// TIA Portal V20 export
// export: Created 2025-12-01T14:57:26.6006718Z, ExportSetting None, DisplayName Totally Integrated Automation Portal, DisplayVersion V20 Update 3, DisplayName TIA Portal Openness, DisplayVersion V20 Update 3, DisplayName TIA Portal Version Control Interface, DisplayVersion V20 Update 3, DisplayName STEP 7 Professional, DisplayVersion V20 Update 3, DisplayName STEP 7 Safety, DisplayVersion V20 Update 2, DisplayName WinCC Basic/Comfort/Advanced, DisplayVersion V20 Update 3, DisplayName WinCC Professional, DisplayVersion V20 Update 3, DisplayName WinCC Unified, DisplayVersion V20 Update 3
FUNCTION "FC601_AJUSTE_SORTER_NEW" : Void   // FC601, LAD
{ S7_Optimized_Access := 'FALSE' }
// stored: AutoNumber false, SetENOAutomatically false
   VAR_INPUT
      Dato_encoder : DInt;
      Detector_referencia : Bool;
      activar_ajuste : Bool;
   END_VAR
   VAR_IN_OUT
      maux_fp_ajuste : Bool;
      maux_fp_detector : Bool;
      primer_flanco : DInt;
      segundo_flanco : DInt;
      tercer_flanco : DInt;
      cuarto_flanco : DInt;
      fin_medicion : Bool;
   END_VAR
   VAR_TEMP   // added for the SCL form of the ladder/FBD networks
      _w1 : Bool;
      _w2 : Bool;
   END_VAR
BEGIN

REGION Network 1
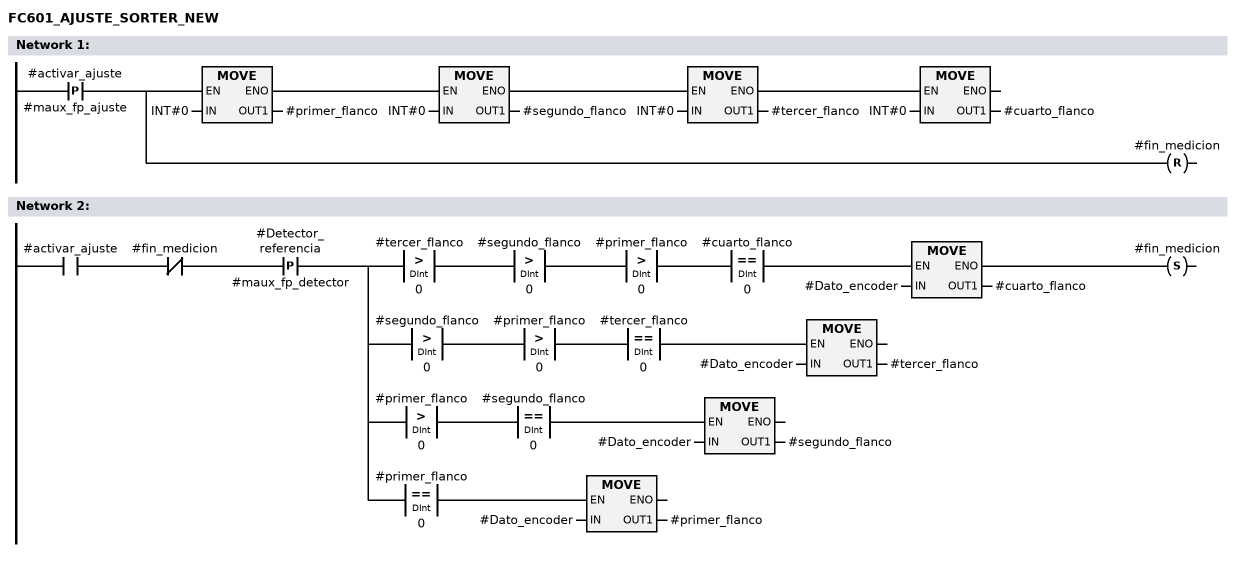
   RUNG wire#powerrail
      P_Contact(operand := #activar_ajuste, bit := #maux_fp_ajuste)
      wire#w1
      { S7_GenerateENO := "TRUE" } Move(in := INT#0, out1 => #primer_flanco)
      { S7_GenerateENO := "TRUE" } Move(in := INT#0, out1 => #segundo_flanco)
      { S7_GenerateENO := "TRUE" } Move(in := INT#0, out1 => #tercer_flanco)
      { S7_GenerateENO := "TRUE" } Move(in := INT#0, out1 => #cuarto_flanco)
   END_RUNG
   RUNG wire#w1
      R_Coil( #fin_medicion )
   END_RUNG
   // the same network as SCL:
   // ENO of a box is taken as its EN; it also drops when the box reports an error
   #_w1 := #activar_ajuste AND NOT #maux_fp_ajuste;   // rising edge of #activar_ajuste
   #maux_fp_ajuste := #activar_ajuste;
   IF #_w1 THEN
       #primer_flanco := INT#0;
       #segundo_flanco := INT#0;
       #tercer_flanco := INT#0;
       #cuarto_flanco := INT#0;
       #fin_medicion := FALSE;
   END_IF;
END_REGION

REGION Network 2
   RUNG wire#powerrail
      Contact( #activar_ajuste )
      I_Contact( #fin_medicion )
      P_Contact(operand := #Detector_referencia, bit := #maux_fp_detector)
      wire#w1
      { S7_Templates := "SrcType := DInt" } GT_Contact(in1 := #tercer_flanco, in2 := 0)
      { S7_Templates := "SrcType := DInt" } GT_Contact(in1 := #segundo_flanco, in2 := 0)
      { S7_Templates := "SrcType := DInt" } GT_Contact(in1 := #primer_flanco, in2 := 0)
      { S7_Templates := "SrcType := DInt" } EQ_Contact(in1 := #cuarto_flanco, in2 := 0)
      Move(in := #Dato_encoder, out1 => #cuarto_flanco)
      S_Coil( #fin_medicion )
   END_RUNG
   RUNG wire#w1
      { S7_Templates := "SrcType := DInt" } GT_Contact(in1 := #segundo_flanco, in2 := 0)
      { S7_Templates := "SrcType := DInt" } GT_Contact(in1 := #primer_flanco, in2 := 0)
      { S7_Templates := "SrcType := DInt" } EQ_Contact(in1 := #tercer_flanco, in2 := 0)
      Move(in := #Dato_encoder, out1 => #tercer_flanco)
   END_RUNG
   RUNG wire#w1
      { S7_Templates := "SrcType := DInt" } GT_Contact(in1 := #primer_flanco, in2 := 0)
      { S7_Templates := "SrcType := DInt" } EQ_Contact(in1 := #segundo_flanco, in2 := 0)
      Move(in := #Dato_encoder, out1 => #segundo_flanco)
   END_RUNG
   RUNG wire#w1
      { S7_Templates := "SrcType := DInt" } EQ_Contact(in1 := #primer_flanco, in2 := 0)
      Move(in := #Dato_encoder, out1 => #primer_flanco)
   END_RUNG
   // the same network as SCL:
   #_w1 := #activar_ajuste AND NOT #fin_medicion AND #Detector_referencia AND NOT #maux_fp_detector;   // rising edge of #Detector_referencia
   #maux_fp_detector := #Detector_referencia;
   #_w2 := #_w1 AND (#tercer_flanco > 0) AND (#segundo_flanco > 0) AND (#primer_flanco > 0) AND (#cuarto_flanco = 0);
   IF #_w2 THEN
       #cuarto_flanco := #Dato_encoder;
       #fin_medicion := TRUE;
   END_IF;
   IF #_w1 AND (#segundo_flanco > 0) AND (#primer_flanco > 0) AND (#tercer_flanco = 0) THEN
       #tercer_flanco := #Dato_encoder;
   END_IF;
   IF #_w1 AND (#primer_flanco > 0) AND (#segundo_flanco = 0) THEN #segundo_flanco := #Dato_encoder; END_IF;
   IF #_w1 AND (#primer_flanco = 0) THEN #primer_flanco := #Dato_encoder; END_IF;
END_REGION
END_FUNCTION
